INTERFACE IOut

PROPERTY Out : LREAL
GET
END_GET
END_PROPERTY

END_INTERFACE

(* stored: Version 1.1.0.1
   Itf IOut: Id {1f5a0544-bc51-4807-af84-0f40e0d77d06}
   Property Out: Id {200fa39f-bcde-49b7-acdb-b61231071a60}
   Get Get: Id {9a0cb42f-bf48-45f2-aee0-dae6a1a41b34} *)
